Staubli VAL3: remSetMaxDist.pgx

program remSetMaxDist(string& sArgs[] (dimensions=1), string& sReturn[] (dimensions=1))
begin
  // Set the maximum allowed move dist in mm
  //
  logMsg("call remSetMaxDist")
  call remSetnGlobal(sArgs,nMaxDist,0,5000,"SETMAXDIST",sReturn)
end
